// TwinCAT 3 PLC project Sample01
// ProgramVersion: 3.1.4024.0
// libraries:
//   Tc2_Standard, * (Beckhoff Automation GmbH)
//   Tc2_System, * (Beckhoff Automation GmbH)
//   Tc3_Module, * (Beckhoff Automation GmbH)
// project tree:
//   / PlcTask.TcTTO
//   POUs/ Class Diagram.TcCD (not stored), FB_Building.TcPOU, FB_Floor.TcPOU, FB_Lamp.TcPOU, FB_Room.TcPOU, F_CalcPowerConsumption.TcPOU, MAIN.TcPOU
// real-time tasks:
//   TASK PlcTask: cycle T#10ms, priority 20, ADS port 350

CONFIGURATION Sample01
    RESOURCE PLC ON TwinCAT3
        TASK PlcTask(INTERVAL := T#10ms, PRIORITY := 20);
        PROGRAM MAIN WITH PlcTask : MAIN;
    END_RESOURCE
END_CONFIGURATION

// ---- POUs/MAIN.TcPOU
PROGRAM MAIN
VAR
	fbBuilding				: FB_Building;
	nPowerConsumption		: UDINT;
	bCalc					: BOOL;
END_VAR

IF (bCalc) THEN
	bCalc := FALSE;
	nPowerConsumption := F_CalcPowerConsumption(fbBuilding);
END_IF

END_PROGRAM

// ---- POUs/FB_Building.TcPOU
FUNCTION_BLOCK FB_Building
VAR_INPUT
END_VAR
VAR_OUTPUT
END_VAR
VAR
	_aFloors	: ARRAY [1..5] OF FB_Floor;
END_VAR

METHOD CalcPowerConsumption : UDINT
VAR
	nFloor		: INT;
END_VAR
FOR nFloor := 1 TO 5 DO
	CalcPowerConsumption := CalcPowerConsumption + refFloors[nFloor].CalcPowerConsumption();
END_FOR
END_METHOD

PROPERTY refFloors : REFERENCE TO ARRAY [1..5] OF FB_Floor
GET
refFloors REF= THIS^._aFloors;
END_GET
END_PROPERTY

END_FUNCTION_BLOCK

// ---- POUs/FB_Floor.TcPOU
FUNCTION_BLOCK FB_Floor
VAR_INPUT
END_VAR
VAR_OUTPUT
END_VAR
VAR
	_aRooms		: ARRAY [1..20] OF FB_Room;
END_VAR

METHOD CalcPowerConsumption : UDINT
VAR
	nRoom		: INT;
END_VAR
FOR nRoom := 1 TO 20 DO	
	CalcPowerConsumption := CalcPowerConsumption + refRooms[nRoom].CalcPowerConsumption();
END_FOR
END_METHOD

PROPERTY refRooms : REFERENCE TO ARRAY [1..20] OF FB_Room
GET
refRooms REF= THIS^._aRooms;
END_GET
END_PROPERTY

END_FUNCTION_BLOCK

// ---- POUs/FB_Room.TcPOU
FUNCTION_BLOCK FB_Room
VAR_INPUT
END_VAR
VAR_OUTPUT
END_VAR
VAR
	_aLamps		: ARRAY [1..10] OF FB_Lamp;
END_VAR

METHOD CalcPowerConsumption : UDINT
VAR_INPUT
END_VAR
VAR
	nLamp		:	INT;
END_VAR
FOR nLamp := 1 TO 10 DO
	CalcPowerConsumption := CalcPowerConsumption + refLamps[nLamp].nPowerConsumption;
END_FOR
END_METHOD

PROPERTY refLamps : REFERENCE TO ARRAY [1..10] OF FB_Lamp
GET
refLamps REF= THIS^._aLamps;
END_GET
END_PROPERTY

END_FUNCTION_BLOCK

// ---- POUs/FB_Lamp.TcPOU
FUNCTION_BLOCK FB_Lamp
VAR_INPUT
END_VAR
VAR_OUTPUT
END_VAR
VAR
	_nPowerConsumption	: UDINT := 1234;
END_VAR

PROPERTY nPowerConsumption : UDINT
GET
nPowerConsumption := _nPowerConsumption;
END_GET
END_PROPERTY

END_FUNCTION_BLOCK

// ---- POUs/F_CalcPowerConsumption.TcPOU
FUNCTION F_CalcPowerConsumption : UDINT
VAR_INPUT
	refBuilding				: REFERENCE TO FB_Building;
END_VAR
VAR
	nFloor, nRoom, nLamp	: INT;
END_VAR

IF (NOT __ISVALIDREF(refBuilding)) THEN
	F_CalcPowerConsumption := 0;
	RETURN;
END_IF

// Violate the Demeter's Law
//FOR nFloor := 1 TO 5 DO
//	FOR nRoom := 1 TO 20 DO
//		FOR nLamp := 1 TO 10 DO
//			F_CalcPowerConsumption := F_CalcPowerConsumption + refBuilding.refFloors[nFloor].refRooms[nRoom].refLamps[nLamp].nPowerConsumption;
//		END_FOR
//	END_FOR
//END_FOR

// Don't violate the Demeter's Law
F_CalcPowerConsumption := refBuilding.CalcPowerConsumption();

END_FUNCTION
